FUNCTION_BLOCK Imwrite (* openCV write image *)
  (* Version 1.0, Alex, SWDC RTSoft *)
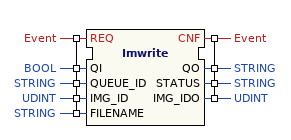
  EVENT_INPUT
    REQ WITH QI, QUEUE_ID, IMG_ID, FILENAME;
  END_EVENT
  EVENT_OUTPUT
    CNF WITH QO, STATUS, IMG_IDO;
  END_EVENT
  VAR_INPUT
    QI : BOOL;
    QUEUE_ID : STRING;
    IMG_ID : UDINT;
    FILENAME : STRING;
  END_VAR
  VAR_OUTPUT
    QO : STRING;
    STATUS : STRING;
    IMG_IDO : UDINT;
  END_VAR
  (* Service APPLICATION/RESOURCE: Service Interface Function Block Type *)
END_FUNCTION_BLOCK
